TYPE TL_BUSY :
(
	eTlBusyStart := 0,
	eTlStartEntranceConveyor,
	eTlStartUpwardsConveyor,
	eTlExecutePalletizer,
	eTlSignalError
)UINT;
END_TYPE

(* stored: Version 1.1.0.1, ProductVersion 3.1.4024.0
   DUT TL_BUSY: Id {196ef372-6d38-4a30-8a23-4e8c520c63ff} *)
